// Brief: Setup Arm Adjust
FUNCTION_BLOCK PUBLIC FB_SetupCtrlAutoAdjust EXTENDS FB_SetupArmCtrlBase
VAR
	// jnt5 adjust velocity
	m_jnt5MaxAdjustVel :LREAL:=3.0*g_deg2Rad;
	m_jnt5MaxAdjustVelWithTrocar :LREAL:=1.0*g_deg2Rad;
	m_jnt5MaxAdjustVelNoTrocar :LREAL:=3.0*g_deg2Rad;
	m_jnt5MaxAdjustAcc :LREAL:=10*g_deg2Rad;
	m_jnt5MaxAdjustJerk :LREAL:=100*g_deg2Rad;
	
	// jnt5 enabled time period
	m_jnt5EnableTime :LREAL :=0;
	
	// time threshold to drive jnt5 after it's enabled
	m_jnt5AdjustWaitTime :LREAL := 0.25;
	
	// traj filter
	m_jnt5TargetPos :LREAL;
	m_jnt5MotionOTG :FB_thirdOrdTrajFilter;
	
END_VAR

// override this function in each exact controller
METHOD PROTECTED calcCmdJntPos : BOOL
VAR_IN_OUT CONSTANT
	i_setupArm	:FB_SetupArm;
END_VAR


VAR 
	i :INT;
END_VAR
IF m_jntEnableFlag[5] = 0 THEN
	RETURN;
END_IF

m_jnt5EnableTime := m_jnt5EnableTime + g_setupArmCtrlCycleTime;

//check trocar single,change control velocity
IF i_setupArm.trocarOn THEN
	m_jnt5MaxAdjustVel := 1.0*g_deg2Rad;
ELSE
	m_jnt5MaxAdjustVel := 3.0*g_deg2Rad;
END_IF
m_jnt5MotionOTG.setMaxV(m_jnt5MaxAdjustVel);

// update command position
IF m_jnt5EnableTime>m_jnt5AdjustWaitTime THEN
	// target joint postion
	IF i_setupArm.jnt5AdjustDir >0 THEN
		m_jnt5TargetPos := GVL_SetupMotorParameters.g_maxJntPos[i_setupArm.armIdx, 5] - g_setupJntPosLimitBuffer[5];
	ELSIF  i_setupArm.jnt5AdjustDir <0 THEN
		m_jnt5TargetPos := GVL_SetupMotorParameters.g_minJntPos[i_setupArm.armIdx, 5] + g_setupJntPosLimitBuffer[5];
	END_IF
	m_jnt5MotionOTG.run(i_targetPos:=m_jnt5TargetPos , i_targetVel:= 0.0, i_targetAcc:= 0.0, o_cmdAcc=> m_cmdJntAcc[5] , o_cmdVel=>m_cmdJntVel[5] , o_cmdPos=>m_cmdJntPos[5]);
END_IF
END_METHOD

METHOD PUBLIC init : BOOL
VAR_IN_OUT CONSTANT
	i_setupArm	:FB_SetupArm;
END_VAR
VAR_IN_OUT 
	r_setupArmCtrlCmd :ST_SetupArmCtrlCmds;
END_VAR
SUPER^.Init(i_setupArm,r_setupArmCtrlCmd);
m_jnt5EnableTime :=0;
m_jnt5MaxAdjustVel :=3.0*g_deg2Rad;
m_jnt5MotionOTG.init(i_curCmdPos:= m_cmdJntPos[5], i_curCmdVel:= 0, i_curCmdAcc:= 0, i_maxV:=m_jnt5MaxAdjustVel , i_maxA:=m_jnt5MaxAdjustAcc, i_maxJ := m_jnt5MaxAdjustJerk, i_Ts:=g_setupArmCtrlCycleTime );
m_jntEnableFlag[5] :=  BOOL_TO_INT( NOT (SafetyCheck.m_SafetyCheck.m_jntErrFlag[i_setupArm.armIdx, 0, 3] OR  SafetyCheck.m_SafetyCheck.m_jntErrFlag[i_setupArm.armIdx, 5, 3]));
END_METHOD

END_FUNCTION_BLOCK

(* stored: Version 1.1.0.1, ProductVersion 3.1.4024.11
   POU FB_SetupCtrlAutoAdjust: Id {53032ea5-b008-491f-a641-5219ef32615c}, SpecialFunc None
   Method calcCmdJntPos: Id {5404c0fa-9750-47fa-bb77-b814ebcded59}
   Method init: Id {d059da11-85f0-484c-8fc1-04c8d016a513} *)
